// TIA Portal project "Trafik Işıkları Uygulaması 2" (V17)

(* hardware
DEVICE "S7-1200 station_1"  S7-1200 Station
   slot 0: "Rack_0"  S7-1200 Rack  Rack  V1.0
   slot 1: "PLC_1"  CPU 1212C AC/DC/Rly  6ES7 212-1BE40-0XB0  V4.4
*)

// ===== PLC "PLC_1"  CPU 1212C AC/DC/Rly =====

VAR_GLOBAL   // PLC tag table "Default tag table"
   "START" AT %E0.0 : Bool;
   "A K, B Y, A YY, B YK" AT %A0.0 : Bool;
   "BAKIM" AT %E0.1 : Bool;
   "YARDIMCI KONTAK" AT %M0.0 : Bool;
   "STOP" AT %I0.2 : Bool;
   "DÖNGÜ" AT %M0.1 : Bool;
   "A YK, A Y, B K, B YY" AT %Q0.1 : Bool;
   "A S, B S" AT %Q0.2 : Bool;
   "BAKIM YARDIMCI KONTAK" AT %M0.2 : Bool;
   "Tag_1" AT %M0.5 : Bool;
   "Tag_2" AT %M0.6 : Bool;
   "Clock_Byte" AT %MB8 : Byte;
   "Clock_10Hz" AT %M8.0 : Bool;
   "Clock_5Hz" AT %M8.1 : Bool;
   "Clock_2.5Hz" AT %M8.2 : Bool;
   "Clock_2Hz" AT %M8.3 : Bool;
   "Clock_1.25Hz" AT %M8.4 : Bool;
   "Clock_1Hz" AT %M8.5 : Bool;
   "Clock_0.625Hz" AT %M8.6 : Bool;
   "Clock_0.5Hz" AT %M8.7 : Bool;
END_VAR

// folder: System blocks/Program resources

DATA_BLOCK "T0"   // DB2
{ S7_Optimized_Access := 'TRUE' }
AUTHOR : Simatic
FAMILY : IEC
NAME : IEC_TMR
VERSION : 1.0
// stored: InstanceOfName IEC_TIMER
"IEC_TIMER"
BEGIN
END_DATA_BLOCK

// folder: (top level)

ORGANIZATION_BLOCK "Main"   // OB1, LAD, ProgramCycle
TITLE = "Main Program Sweep (Cycle)"
{ S7_Optimized_Access := 'TRUE' }
VERSION : 0.1
   VAR_INPUT
      Initial_Call : Bool;   // Initial call of this OB
      Remanence : Bool;   // =True, if remanent data are available
   END_VAR
BEGIN

REGION Network 1
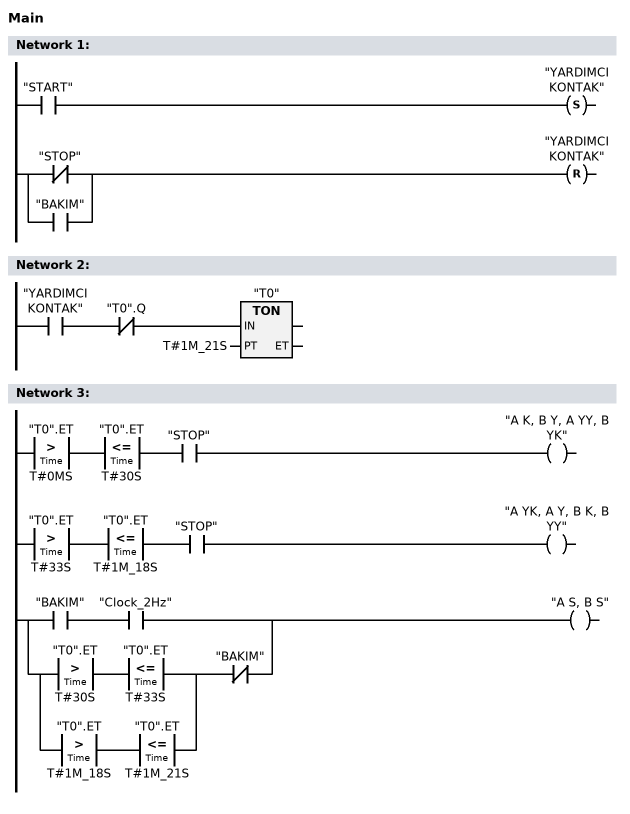
   RUNG wire#powerrail
      Contact( "START" )
      S_Coil( "YARDIMCI KONTAK" )
   END_RUNG
   RUNG wire#powerrail
      I_Contact( "STOP" )
      wire#w1
      R_Coil( "YARDIMCI KONTAK" )
   END_RUNG
   RUNG wire#powerrail
      Contact( "BAKIM" )
   END_RUNG wire#w1
   // the same network as SCL:
   IF "START" THEN "YARDIMCI KONTAK" := TRUE; END_IF;
   IF NOT "STOP" OR "BAKIM" THEN "YARDIMCI KONTAK" := FALSE; END_IF;
END_REGION

REGION Network 2
   "T0".TON(IN := "YARDIMCI KONTAK" AND NOT "T0".Q, PT := T#1M_21S);
END_REGION

REGION Network 3
   RUNG wire#powerrail
      { S7_Templates := "SrcType := Time" } GT_Contact(in1 := "T0".ET, in2 := T#0MS)
      { S7_Templates := "SrcType := Time" } LE_Contact(in1 := "T0".ET, in2 := T#30S)
      Contact( "STOP" )
      Coil( "A K, B Y, A YY, B YK" )
   END_RUNG
   RUNG wire#powerrail
      { S7_Templates := "SrcType := Time" } GT_Contact(in1 := "T0".ET, in2 := T#33S)
      { S7_Templates := "SrcType := Time" } LE_Contact(in1 := "T0".ET, in2 := T#1M_18S)
      Contact( "STOP" )
      Coil( "A YK, A Y, B K, B YY" )
   END_RUNG
   RUNG wire#powerrail
      Contact( "BAKIM" )
      Contact( "Clock_2Hz" )
      wire#w1
      Coil( "A S, B S" )
   END_RUNG
   RUNG wire#powerrail
      { S7_Templates := "SrcType := Time" } GT_Contact(in1 := "T0".ET, in2 := T#30S)
      { S7_Templates := "SrcType := Time" } LE_Contact(in1 := "T0".ET, in2 := T#33S)
      wire#w2
      I_Contact( "BAKIM" )
   END_RUNG wire#w1
   RUNG wire#powerrail
      { S7_Templates := "SrcType := Time" } GT_Contact(in1 := "T0".ET, in2 := T#1M_18S)
      { S7_Templates := "SrcType := Time" } LE_Contact(in1 := "T0".ET, in2 := T#1M_21S)
   END_RUNG wire#w2
   // the same network as SCL:
   "A K, B Y, A YY, B YK" := ("T0".ET > T#0MS) AND ("T0".ET <= T#30S) AND "STOP";
   "A YK, A Y, B K, B YY" := ("T0".ET > T#33S) AND ("T0".ET <= T#1M_18S) AND "STOP";
   "A S, B S" := ("BAKIM" AND "Clock_2Hz") OR (((("T0".ET > T#30S) AND ("T0".ET <= T#33S)) OR (("T0".ET > T#1M_18S) AND ("T0".ET <= T#1M_21S))) AND NOT "BAKIM");
END_REGION
END_ORGANIZATION_BLOCK